// TIA Portal V19 export
// export: Created 2024-12-05T09:06:09.6853574Z, ExportSetting WithDefaults, DisplayName Totally Integrated Automation Portal, DisplayVersion V19 Update 1, DisplayName TIA Portal Openness, DisplayVersion V19 Update 1, DisplayName TIA Portal Version Control Interface, DisplayVersion V19, DisplayName SINAMICS Startdrive Advanced, DisplayVersion V19, DisplayName SINAMICS DCC, DisplayVersion V19, DisplayName SINAMICS Startdrive G130, G150, S120, S150, SINAMICS MV, G220, S200, S210, DisplayVersion V19, DisplayName SINAMICS Startdrive G110M, G120, G120C, G120D, G120P, G115D, DisplayVersion V19, DisplayName STEP 7 Professional, DisplayVersion V19 Update 1, DisplayName STEP 7 Safety, DisplayVersion V19 Update 1, DisplayName WinCC Advanced, DisplayVersion V19 Update 1, DisplayName WinCC Advanced / Unified PC, DisplayVersion V19 Update 1
DATA_BLOCK "GLOBAL"   // DB9
{ S7_Optimized_Access := 'TRUE' }
VERSION : 0.1
// stored: AutoNumber true, DBAccessibleFromOPCUA true, DBAccessibleFromWebserver true, InstanceOfName EM_GLOBAL, InstanceOfType UDT, IsOnlyStoredInLoadMemory false, IsWriteProtectedInAS false
"EM_GLOBAL"
   // VAR
   //    Gen : "GLOBAL_Gen";
   //    Param : "GLOBAL_Param";
   //    Recipe : "GLOBAL_Recipe";
   //    AlmLong : "GLOBAL_Alm";
   //    AlmTypeFbkLong : "AlmType";
   //    AlmTypeOkLong : "AlmType";
   //    AlmCauseFbkLong : "AlmCause";
   //    AlmCauseOkLong : "AlmCause";
   //    AlmStructLong : "STD_ALM_STRUCT";
   //    AlmBannerFbkLong : "STD_ALM_BAN_FBK";
   //    AlmShort : "GLOBAL_Alm";
   //    AlmTypeFbkShort : "AlmType";
   //    AlmTypeOkShort : "AlmType";
   //    AlmCauseFbkShort : "AlmCause";
   //    AlmCauseOkShort : "AlmCause";
   //    AlmStructShort : "STD_ALM_STRUCT";
   //    AlmBannerFbkShort : "STD_ALM_BAN_FBK";
   //    Sign : "GLOBAL_Sign";
   //    SignStruct : "STD_SIGN_STRUCT";
   //    SignBannerFbk : "STD_SIGN_BAN_FBK";
   //    Input : "GLOBAL_Input";
   //    Output : "GLOBAL_Output";
   //    Ons : "GLOBAL_Ons";
   //    AirTreatment : "AirTreatment";
   //    Summ : "GLOBAL_Summary";
   //    LightSiren : "LightSiren_Module";
   //    ExchangeCmd : "Exchange_FromGlobal";
   //    ExchangeCmd_Switchboard : "Exchange_FromGlobal_Switchboard";
   //    Downstream : "Interface_Downstream";
   //    "MyStateDeviceCab&Field" : Array[0..1023] of Bool;
   //    DC_Bus_Converter1 : "ACT_DC_BUS";
   //    DC_Bus_Converter2 : "ACT_DC_BUS";
   //    DC_Bus_Converter3 : "ACT_DC_BUS";
   //    DC_Bus_Converter4 : "ACT_DC_BUS";
   // END_VAR
BEGIN
   Gen.PlannerGroupSync := TRUE;
   Gen.PwrDriveShortCondOK := TRUE;
   Gen.PwrDriveLongCondOK := TRUE;
   Gen.PwrDriveShortDone := TRUE;
   Gen.PwrDriveLongDone := TRUE;
   Gen.StationOutOfTime := TRUE;
   Gen.AllPlcsRun := TRUE;
   Gen.PwrDriveShortIndex := 8192;
   Gen.PwrDriveLongIndex := 8192;
   Gen.DayOfWeek := 5;
   Gen.PanelConnectionError := 64;
   Gen.FirstAlmID := -1;
   Gen.TimePIDexecution := 8.0;
   Gen.TON_ResetNewAlm.PT := T#5S;
   Gen.TON_ResetNewSign.PT := T#1S;
   Gen.TON_PlannerGroupSync.PT := T#2S;
   Gen.TON_PlannerGroupSync.ET := T#2S;
   Gen.TON_PlannerGroupSync.IN := TRUE;
   Gen.TON_PlannerGroupSync.Q := TRUE;
   Gen.TON_WaitSaveRecipeOnLine.PT := T#5S;
   Gen.TON_WaitLoadRecipeOnLine.PT := T#5S;
   Gen.TON_AirMissing_Gta1.PT := T#2S;
   Gen.TON_AirMissing_Gta2.PT := T#2S;
   Gen.TON_AirMissing_Gta3.PT := T#2S;
   Gen.TON_AirMissing_Gta4.PT := T#2S;
   Gen.TON_AirMissing_Gta4.ET := T#2S;
   Gen.TON_AirMissing_Gta4.IN := TRUE;
   Gen.TON_AirMissing_Gta4.Q := TRUE;
   Gen.TON_AirMissing_Gta5.PT := T#2S;
   Gen.TON_AirMissing_Gta5.ET := T#2S;
   Gen.TON_AirMissing_Gta5.IN := TRUE;
   Gen.TON_AirMissing_Gta5.Q := TRUE;
   Gen.TON_AirMissing_Gta6.PT := T#2S;
   Gen.TON_RecipeDownloadTimeout.PT := T#5S;
   Gen.TON_RecipeUploadTimeout.PT := T#5S;
   Gen.TON_RecipeMaintConfigDownloadTimeout.PT := T#5S;
   Gen.TON_RecipeMaintConfigUploadTimeout.PT := T#5S;
   Gen.TON_RecipeTotalizersDownloadTimeout.PT := T#5S;
   Gen.TON_RecipeTotalizersUploadTimeout.PT := T#5S;
   Gen.TOF_ResetButtonAuto.PT := T#1S;
   Gen.TOF_ResetButtonAuto.ET := T#1S;
   Gen.TOF_ResetButtonGlobal.PT := T#300MS;
   Gen.TOF_ResetButtonGlobal.ET := T#300MS;
   Gen.TOF_SirenEna.PT := T#5S;
   Gen.TOF_SirenEna.ET := T#5S;
   Gen.TON_LineEmpty.PT := T#2S;
   Recipe.MngByHmi := TRUE;
   Recipe.MaxNumber := 99;
   Recipe.Online.TOF_SaveDone.PT := T#1S;
   Recipe.Online.TOF_LoadDone.PT := T#1S;
   Recipe.Offline.TOF_SaveDone.PT := T#1S;
   Recipe.Offline.TOF_LoadDone.PT := T#1S;
   // AlmLong.ThSwitch."0" : GLOBAL.AlmLong.ThSwitch.0 > Circuit breaker power supply 1 (1PW100QA8)
   // AlmLong.ThSwitch."1" : GLOBAL.AlmLong.ThSwitch.1 > Circuit breaker power supply 2 (1PW100QA9)
   // AlmLong.ThSwitch."2" : GLOBAL.AlmLong.ThSwitch.2 > Circuit breaker series main power supply (1PW113)
   // AlmLong.ThSwitch."3" : GLOBAL.AlmLong.ThSwitch.3 > Circuit breaker series field power supply (1PW114)
   // AlmLong.ThSwitch."4" : GLOBAL.AlmLong.ThSwitch.4 > Circuit breaker series sinamics power supply (1PW113)
   // AlmLong.ThSwitch."5" : GLOBAL.AlmLong.ThSwitch.5 > Circuit breaker series valves power supply (1PW116)
   // AlmLong.ThSwitch."6" : GLOBAL.AlmLong.ThSwitch.6 > Circuit breaker series lamps power supply (1PW115)
   // AlmLong.ThSwitch."7" : GLOBAL.AlmLong.ThSwitch.7 > Main trip isolator unit faul (1PW6KA2)
   // AlmLong.ThSwitch."8" : GLOBAL.AlmLong.ThSwitch.8
   // AlmLong.ThSwitch."9" : GLOBAL.AlmLong.ThSwitch.9
   // AlmLong.ThSwitch."10" : GLOBAL.AlmLong.ThSwitch.10 > Circuit breaker series blocking cycle (1PW110)
   // AlmLong.ThSwitch."11" : GLOBAL.AlmLong.ThSwitch.11 > Loto disconnected (1PW11QA2)
   // AlmLong.ThSwitch."12" : GLOBAL.AlmLong.ThSwitch.12
   // AlmLong.ThSwitch."13" : GLOBAL.AlmLong.ThSwitch.13 > Circuit breakers series depositors (1PW110)
   // AlmLong.ThSwitch."14" : GLOBAL.AlmLong.ThSwitch.14
   // AlmLong.ThSwitch."15" : GLOBAL.AlmLong.ThSwitch.15
   // AlmLong.ThSwitch."16" : GLOBAL.AlmLong.ThSwitch.16
   // AlmLong.ThSwitch."17" : GLOBAL.AlmLong.ThSwitch.17
   // AlmLong.ThSwitch."18" : GLOBAL.AlmLong.ThSwitch.18
   // AlmLong.ThSwitch."19" : GLOBAL.AlmLong.ThSwitch.19
   // AlmLong.ThSwitch."20" : GLOBAL.AlmLong.ThSwitch.20
   // AlmLong.ThSwitch."21" : GLOBAL.AlmLong.ThSwitch.21
   // AlmLong.ThSwitch."22" : GLOBAL.AlmLong.ThSwitch.22
   // AlmLong.ThSwitch."23" : GLOBAL.AlmLong.ThSwitch.23
   // AlmLong.ThSwitch."24" : GLOBAL.AlmLong.ThSwitch.24
   // AlmLong.ThSwitch."25" : GLOBAL.AlmLong.ThSwitch.25
   // AlmLong.ThSwitch."26" : GLOBAL.AlmLong.ThSwitch.26
   // AlmLong.ThSwitch."27" : GLOBAL.AlmLong.ThSwitch.27
   // AlmLong.ThSwitch."28" : GLOBAL.AlmLong.ThSwitch.28
   // AlmLong.ThSwitch."29" : GLOBAL.AlmLong.ThSwitch.29
   // AlmLong.ThSwitch."30" : GLOBAL.AlmLong.ThSwitch.30
   // AlmLong.ThSwitch."31" : GLOBAL.AlmLong.ThSwitch.31
   // AlmLong.SafeComm."0" : GLOBAL.AlmLong.SafeComm.0
   // AlmLong.SafeComm."1" : GLOBAL.AlmLong.SafeComm.1
   // AlmLong.SafeComm."2" : GLOBAL.AlmLong.SafeComm.2 > Fault on ethernet module (1PLC200KF4)
   // AlmLong.SafeComm."3" : GLOBAL.AlmLong.SafeComm.3 > Fault on ethernet module (1PLC200KF4A)
   // AlmLong.SafeComm."4" : GLOBAL.AlmLong.SafeComm.4 > Fault on ethernet module (1PLC200KF5)
   // AlmLong.SafeComm."5" : GLOBAL.AlmLong.SafeComm.5
   // AlmLong.SafeComm."6" : GLOBAL.AlmLong.SafeComm.6
   // AlmLong.SafeComm."7" : GLOBAL.AlmLong.SafeComm.7 > Communication fault DP1
   // AlmLong.SafeComm."8" : GLOBAL.AlmLong.SafeComm.8 > Communication fault DP2
   // AlmLong.SafeComm."9" : GLOBAL.AlmLong.SafeComm.9 > Communication fault DP3
   // AlmLong.SafeComm."10" : GLOBAL.AlmLong.SafeComm.10 > Communication fault DP4
   // AlmLong.SafeComm."11" : GLOBAL.AlmLong.SafeComm.11
   // AlmLong.SafeComm."12" : GLOBAL.AlmLong.SafeComm.12
   // AlmLong.SafeComm."13" : GLOBAL.AlmLong.SafeComm.13
   // AlmLong.SafeComm."14" : GLOBAL.AlmLong.SafeComm.14
   // AlmLong.SafeComm."15" : GLOBAL.AlmLong.SafeComm.15 > Communication fault point_IO 1 (1PLC300KF3)
   // AlmLong.SafeComm."16" : GLOBAL.AlmLong.SafeComm.16 > Communication fault point_IO 2 (1PLC350KF3)
   // AlmLong.SafeComm."17" : GLOBAL.AlmLong.SafeComm.17 > Communication fault point_IO 3 (1PLC400KF3)
   // AlmLong.SafeComm."18" : GLOBAL.AlmLong.SafeComm.18
   // AlmLong.SafeComm."19" : GLOBAL.AlmLong.SafeComm.19
   // AlmLong.SafeComm."20" : GLOBAL.AlmLong.SafeComm.20
   // AlmLong.SafeComm."21" : GLOBAL.AlmLong.SafeComm.21
   // AlmLong.SafeComm."22" : GLOBAL.AlmLong.SafeComm.22
   // AlmLong.SafeComm."23" : GLOBAL.AlmLong.SafeComm.23
   // AlmLong.SafeComm."24" : GLOBAL.AlmLong.SafeComm.24
   // AlmLong.SafeComm."25" : GLOBAL.AlmLong.SafeComm.25
   // AlmLong.SafeComm."26" : GLOBAL.AlmLong.SafeComm.26
   // AlmLong.SafeComm."27" : GLOBAL.AlmLong.SafeComm.27
   // AlmLong.SafeComm."28" : GLOBAL.AlmLong.SafeComm.28
   // AlmLong.SafeComm."29" : GLOBAL.AlmLong.SafeComm.29
   // AlmLong.SafeComm."30" : GLOBAL.AlmLong.SafeComm.30
   // AlmLong.SafeComm."31" : GLOBAL.AlmLong.SafeComm.31
   // AlmLong.SafeEmg."0" : GLOBAL.AlmLong.SafeEmg.0 > Emergency pressed on cabinet (1PLC340SF2)
   // AlmLong.SafeEmg."1" : GLOBAL.AlmLong.SafeEmg.1
   // AlmLong.SafeEmg."2" : GLOBAL.AlmLong.SafeEmg.2
   // AlmLong.SafeEmg."3" : GLOBAL.AlmLong.SafeEmg.3
   // AlmLong.SafeEmg."4" : GLOBAL.AlmLong.SafeEmg.4
   // AlmLong.SafeEmg."5" : GLOBAL.AlmLong.SafeEmg.5
   // AlmLong.SafeEmg."6" : GLOBAL.AlmLong.SafeEmg.6
   // AlmLong.SafeEmg."7" : GLOBAL.AlmLong.SafeEmg.7
   // AlmLong.SafeEmg."8" : GLOBAL.AlmLong.SafeEmg.8
   // AlmLong.SafeEmg."9" : GLOBAL.AlmLong.SafeEmg.9
   // AlmLong.SafeEmg."10" : GLOBAL.AlmLong.SafeEmg.10
   // AlmLong.SafeEmg."11" : GLOBAL.AlmLong.SafeEmg.11
   // AlmLong.SafeEmg."12" : GLOBAL.AlmLong.SafeEmg.12
   // AlmLong.SafeEmg."13" : GLOBAL.AlmLong.SafeEmg.13
   // AlmLong.SafeEmg."14" : GLOBAL.AlmLong.SafeEmg.14
   // AlmLong.SafeEmg."15" : GLOBAL.AlmLong.SafeEmg.15
   // AlmLong.SafeEmg."16" : GLOBAL.AlmLong.SafeEmg.16 > Instruction fault emergency pressed on cabinet (1PLC340SF2)
   // AlmLong.SafeEmg."17" : GLOBAL.AlmLong.SafeEmg.17
   // AlmLong.SafeEmg."18" : GLOBAL.AlmLong.SafeEmg.18
   // AlmLong.SafeEmg."19" : GLOBAL.AlmLong.SafeEmg.19
   // AlmLong.SafeEmg."20" : GLOBAL.AlmLong.SafeEmg.20
   // AlmLong.SafeEmg."21" : GLOBAL.AlmLong.SafeEmg.21
   // AlmLong.SafeEmg."22" : GLOBAL.AlmLong.SafeEmg.22
   // AlmLong.SafeEmg."23" : GLOBAL.AlmLong.SafeEmg.23
   // AlmLong.SafeEmg."24" : GLOBAL.AlmLong.SafeEmg.24
   // AlmLong.SafeEmg."25" : GLOBAL.AlmLong.SafeEmg.25
   // AlmLong.SafeEmg."26" : GLOBAL.AlmLong.SafeEmg.26
   // AlmLong.SafeEmg."27" : GLOBAL.AlmLong.SafeEmg.27
   // AlmLong.SafeEmg."28" : GLOBAL.AlmLong.SafeEmg.28
   // AlmLong.SafeEmg."29" : GLOBAL.AlmLong.SafeEmg.29
   // AlmLong.SafeEmg."30" : GLOBAL.AlmLong.SafeEmg.30
   // AlmLong.SafeEmg."31" : GLOBAL.AlmLong.SafeEmg.31 > Moulding emergency series safety no ok
   // AlmLong.SafeGuards."0" : GLOBAL.AlmLong.SafeGuards.0
   // AlmLong.SafeGuards."1" : GLOBAL.AlmLong.SafeGuards.1
   // AlmLong.SafeGuards."2" : GLOBAL.AlmLong.SafeGuards.2
   // AlmLong.SafeGuards."3" : GLOBAL.AlmLong.SafeGuards.3
   // AlmLong.SafeGuards."4" : GLOBAL.AlmLong.SafeGuards.4
   // AlmLong.SafeGuards."5" : GLOBAL.AlmLong.SafeGuards.5
   // AlmLong.SafeGuards."6" : GLOBAL.AlmLong.SafeGuards.6
   // AlmLong.SafeGuards."7" : GLOBAL.AlmLong.SafeGuards.7
   // AlmLong.SafeGuards."8" : GLOBAL.AlmLong.SafeGuards.8
   // AlmLong.SafeGuards."9" : GLOBAL.AlmLong.SafeGuards.9
   // AlmLong.SafeGuards."10" : GLOBAL.AlmLong.SafeGuards.10
   // AlmLong.SafeGuards."11" : GLOBAL.AlmLong.SafeGuards.11
   // AlmLong.SafeGuards."12" : GLOBAL.AlmLong.SafeGuards.12
   // AlmLong.SafeGuards."13" : GLOBAL.AlmLong.SafeGuards.13
   // AlmLong.SafeGuards."14" : GLOBAL.AlmLong.SafeGuards.14
   // AlmLong.SafeGuards."15" : GLOBAL.AlmLong.SafeGuards.15
   // AlmLong.SafeGuards."16" : GLOBAL.AlmLong.SafeGuards.16 > Module fault (1PLC340KF1)
   // AlmLong.SafeGuards."17" : GLOBAL.AlmLong.SafeGuards.17 > Module fault (1PLC390KF1)
   // AlmLong.SafeGuards."18" : GLOBAL.AlmLong.SafeGuards.18 > Module fault (1PLC391KF1)
   // AlmLong.SafeGuards."19" : GLOBAL.AlmLong.SafeGuards.19 > Module fault (1PLC396KF1)
   // AlmLong.SafeGuards."20" : GLOBAL.AlmLong.SafeGuards.20 > Module fault (1PLC398KF1)
   // AlmLong.SafeGuards."21" : GLOBAL.AlmLong.SafeGuards.21
   // AlmLong.SafeGuards."22" : GLOBAL.AlmLong.SafeGuards.22
   // AlmLong.SafeGuards."23" : GLOBAL.AlmLong.SafeGuards.23
   // AlmLong.SafeGuards."24" : GLOBAL.AlmLong.SafeGuards.24
   // AlmLong.SafeGuards."25" : GLOBAL.AlmLong.SafeGuards.25
   // AlmLong.SafeGuards."26" : GLOBAL.AlmLong.SafeGuards.26
   // AlmLong.SafeGuards."27" : GLOBAL.AlmLong.SafeGuards.27
   // AlmLong.SafeGuards."28" : GLOBAL.AlmLong.SafeGuards.28
   // AlmLong.SafeGuards."29" : GLOBAL.AlmLong.SafeGuards.29
   // AlmLong.SafeGuards."30" : GLOBAL.AlmLong.SafeGuards.30
   // AlmLong.SafeGuards."31" : GLOBAL.AlmLong.SafeGuards.31
   // AlmLong.GtaAirGroup."0" : GLOBAL.AlmLong.GtaAirGroup.0 > Module or instruction fault GTA air group 1 (1FM371BP2,3)
   AlmLong.GtaAirGroup."1" := FALSE;   // GLOBAL.AlmLong.GtaAirGroup.1 > Group GTA 1 missing air (1FM330BP6)
   // AlmLong.GtaAirGroup."2" : GLOBAL.AlmLong.GtaAirGroup.2 > Module or instruction fault GTA air group 2 (3VV372BP2,3)
   // AlmLong.GtaAirGroup."3" : GLOBAL.AlmLong.GtaAirGroup.3 > Group GTA 2 missing air (3VV330BP5)
   // AlmLong.GtaAirGroup."4" : GLOBAL.AlmLong.GtaAirGroup.4 > Module or instruction fault GTA air group 3 (4VV372BP2,3)
   AlmLong.GtaAirGroup."5" := FALSE;   // GLOBAL.AlmLong.GtaAirGroup.5 > Group GTA 3 missing air (4VV330BP5)
   AlmLong.GtaAirGroup."6" := TRUE;   // GLOBAL.AlmLong.GtaAirGroup.6 > Module or instruction fault GTA air group 4 (1RD372BP2,3)
   AlmLong.GtaAirGroup."7" := TRUE;   // GLOBAL.AlmLong.GtaAirGroup.7 > Group GTA 4 missing air (1RD330BP5)
   // AlmLong.GtaAirGroup."8" : GLOBAL.AlmLong.GtaAirGroup.8 > Module or instruction fault GTA air group 5 (1RD472BP2,3)
   AlmLong.GtaAirGroup."9" := TRUE;   // GLOBAL.AlmLong.GtaAirGroup.9 > Group GTA 5 missing air (1RD430BP2)
   // AlmLong.GtaAirGroup."10" : GLOBAL.AlmLong.GtaAirGroup.10
   // AlmLong.GtaAirGroup."11" : GLOBAL.AlmLong.GtaAirGroup.11
   // AlmLong.GtaAirGroup."12" : GLOBAL.AlmLong.GtaAirGroup.12
   // AlmLong.GtaAirGroup."13" : GLOBAL.AlmLong.GtaAirGroup.13
   // AlmLong.GtaAirGroup."14" : GLOBAL.AlmLong.GtaAirGroup.14
   // AlmLong.GtaAirGroup."15" : GLOBAL.AlmLong.GtaAirGroup.15
   // AlmLong.GtaAirGroup."16" : GLOBAL.AlmLong.GtaAirGroup.16
   // AlmLong.GtaAirGroup."17" : GLOBAL.AlmLong.GtaAirGroup.17
   // AlmLong.GtaAirGroup."18" : GLOBAL.AlmLong.GtaAirGroup.18
   // AlmLong.GtaAirGroup."19" : GLOBAL.AlmLong.GtaAirGroup.19
   // AlmLong.GtaAirGroup."20" : GLOBAL.AlmLong.GtaAirGroup.20
   // AlmLong.GtaAirGroup."21" : GLOBAL.AlmLong.GtaAirGroup.21
   // AlmLong.GtaAirGroup."22" : GLOBAL.AlmLong.GtaAirGroup.22
   // AlmLong.GtaAirGroup."23" : GLOBAL.AlmLong.GtaAirGroup.23
   // AlmLong.GtaAirGroup."24" : GLOBAL.AlmLong.GtaAirGroup.24
   // AlmLong.GtaAirGroup."25" : GLOBAL.AlmLong.GtaAirGroup.25
   // AlmLong.GtaAirGroup."26" : GLOBAL.AlmLong.GtaAirGroup.26
   // AlmLong.GtaAirGroup."27" : GLOBAL.AlmLong.GtaAirGroup.27
   // AlmLong.GtaAirGroup."28" : GLOBAL.AlmLong.GtaAirGroup.28
   // AlmLong.GtaAirGroup."29" : GLOBAL.AlmLong.GtaAirGroup.29
   // AlmLong.GtaAirGroup."30" : GLOBAL.AlmLong.GtaAirGroup.30
   // AlmLong.GtaAirGroup."31" : GLOBAL.AlmLong.GtaAirGroup.31
   // AlmLong.Major."0" : GLOBAL.AlmLong.Major.0 > Module or instruction fault emergency + carter feedback (1CH130KF2)
   // AlmLong.Major."1" : GLOBAL.AlmLong.Major.1 > Module or instruction fault feedback emergency (1CH130KF4)
   // AlmLong.Major."2" : GLOBAL.AlmLong.Major.2 > Module or instruction fault feedback emergency (1CH130KF6)
   // AlmLong.Major."3" : GLOBAL.AlmLong.Major.3 > Module or instruction fault feedback fans emergency contactor branch 2
   // AlmLong.Major."4" : GLOBAL.AlmLong.Major.4
   // AlmLong.Major."5" : GLOBAL.AlmLong.Major.5 > Module or instruction fault feedback emergency + carter branch 1 (1CH132KF2)
   // AlmLong.Major."6" : GLOBAL.AlmLong.Major.6 > Module or instruction fault feedback emergency + carter branch 2 (1CH132KF4)
   // AlmLong.Major."7" : GLOBAL.AlmLong.Major.7
   // AlmLong.Major."8" : GLOBAL.AlmLong.Major.8
   // AlmLong.Major."9" : GLOBAL.AlmLong.Major.9
   // AlmLong.Major."10" : GLOBAL.AlmLong.Major.10
   // AlmLong.Major."11" : GLOBAL.AlmLong.Major.11
   // AlmLong.Major."12" : GLOBAL.AlmLong.Major.12
   // AlmLong.Major."13" : GLOBAL.AlmLong.Major.13
   // AlmLong.Major."14" : GLOBAL.AlmLong.Major.14
   // AlmLong.Major."15" : GLOBAL.AlmLong.Major.15 > Presence 24Vdc supply
   // AlmLong.Major."16" : GLOBAL.AlmLong.Major.16
   // AlmLong.Major."17" : GLOBAL.AlmLong.Major.17
   // AlmLong.Major."18" : GLOBAL.AlmLong.Major.18
   // AlmLong.Major."19" : GLOBAL.AlmLong.Major.19
   // AlmLong.Major."20" : GLOBAL.AlmLong.Major.20 > Dc bus converter 1 fault
   // AlmLong.Major."21" : GLOBAL.AlmLong.Major.21 > Dc bus converter 2 fault
   // AlmLong.Major."22" : GLOBAL.AlmLong.Major.22 > Dc bus converter 3 fault
   // AlmLong.Major."23" : GLOBAL.AlmLong.Major.23 > Dc bus converter 4 fault
   // AlmLong.Major."24" : GLOBAL.AlmLong.Major.24
   // AlmLong.Major."25" : GLOBAL.AlmLong.Major.25
   // AlmLong.Major."26" : GLOBAL.AlmLong.Major.26
   // AlmLong.Major."27" : GLOBAL.AlmLong.Major.27
   // AlmLong.Major."28" : GLOBAL.AlmLong.Major.28
   // AlmLong.Major."29" : GLOBAL.AlmLong.Major.29
   // AlmLong.Major."30" : GLOBAL.AlmLong.Major.30
   // AlmLong.Major."31" : GLOBAL.AlmLong.Major.31
   // AlmLong.Minor."0" : GLOBAL.AlmLong.Minor.0 > Connection HMI server error
   // AlmLong.Minor."1" : GLOBAL.AlmLong.Minor.1 > Request update parameters from PLC to HMI
   // AlmLong.Minor."2" : GLOBAL.AlmLong.Minor.2 > Recipe download from HMI error
   // AlmLong.Minor."3" : GLOBAL.AlmLong.Minor.3 > Request maintenance configuration from PLC to HMI
   // AlmLong.Minor."4" : GLOBAL.AlmLong.Minor.4 > Recipe maintenance configuration download from HMI error
   // AlmLong.Minor."5" : GLOBAL.AlmLong.Minor.5 > Request update totalizers from PLC to HMI
   // AlmLong.Minor."6" : GLOBAL.AlmLong.Minor.6 > Recipe totalizers download from HMI error
   // AlmLong.Minor."7" : GLOBAL.AlmLong.Minor.7
   // AlmLong.Minor."8" : GLOBAL.AlmLong.Minor.8 > More then one drum enabled, they will be reset
   // AlmLong.Minor."9" : GLOBAL.AlmLong.Minor.9
   // AlmLong.Minor."10" : GLOBAL.AlmLong.Minor.10
   // AlmLong.Minor."11" : GLOBAL.AlmLong.Minor.11
   // AlmLong.Minor."12" : GLOBAL.AlmLong.Minor.12
   // AlmLong.Minor."13" : GLOBAL.AlmLong.Minor.13
   // AlmLong.Minor."14" : GLOBAL.AlmLong.Minor.14
   // AlmLong.Minor."15" : GLOBAL.AlmLong.Minor.15 > Downstream communication fault
   // AlmLong.Minor."16" : GLOBAL.AlmLong.Minor.16
   // AlmLong.Minor."17" : GLOBAL.AlmLong.Minor.17
   // AlmLong.Minor."18" : GLOBAL.AlmLong.Minor.18
   // AlmLong.Minor."19" : GLOBAL.AlmLong.Minor.19
   // AlmLong.Minor."20" : GLOBAL.AlmLong.Minor.20
   // AlmLong.Minor."21" : GLOBAL.AlmLong.Minor.21
   // AlmLong.Minor."22" : GLOBAL.AlmLong.Minor.22
   // AlmLong.Minor."23" : GLOBAL.AlmLong.Minor.23
   // AlmLong.Minor."24" : GLOBAL.AlmLong.Minor.24
   // AlmLong.Minor."25" : GLOBAL.AlmLong.Minor.25
   // AlmLong.Minor."26" : GLOBAL.AlmLong.Minor.26
   // AlmLong.Minor."27" : GLOBAL.AlmLong.Minor.27
   // AlmLong.Minor."28" : GLOBAL.AlmLong.Minor.28
   // AlmLong.Minor."29" : GLOBAL.AlmLong.Minor.29
   // AlmLong.Minor."30" : GLOBAL.AlmLong.Minor.30
   // AlmLong.Minor."31" : GLOBAL.AlmLong.Minor.31
   AlmTypeFbkLong.GtaAirGroup := TRUE;
   AlmTypeOkLong.ThSwitch := TRUE;
   AlmTypeOkLong.SafeComm := TRUE;
   AlmTypeOkLong.SafeEmg := TRUE;
   AlmTypeOkLong.SafeGuards := TRUE;
   AlmTypeOkLong.GtaAirGroup := FALSE;
   AlmTypeOkLong.Major := TRUE;
   AlmTypeOkLong.Minor := TRUE;
   AlmTypeOkLong.Spare07 := TRUE;
   AlmTypeOkLong.Spare08 := TRUE;
   AlmTypeOkLong.Spare09 := TRUE;
   AlmTypeOkLong.Spare10 := TRUE;
   AlmTypeOkLong.Spare11 := TRUE;
   AlmTypeOkLong.Spare12 := TRUE;
   AlmTypeOkLong.Spare13 := TRUE;
   AlmTypeOkLong.Spare14 := TRUE;
   AlmTypeOkLong.Spare15 := TRUE;
   AlmTypeOkLong.Spare16 := TRUE;
   AlmTypeOkLong.Spare17 := TRUE;
   AlmTypeOkLong.Spare18 := TRUE;
   AlmTypeOkLong.Spare19 := TRUE;
   AlmTypeOkLong.Spare20 := TRUE;
   AlmTypeOkLong.Spare21 := TRUE;
   AlmTypeOkLong.Spare22 := TRUE;
   AlmTypeOkLong.Spare23 := TRUE;
   AlmTypeOkLong.Spare24 := TRUE;
   AlmTypeOkLong.Spare25 := TRUE;
   AlmTypeOkLong.Spare26 := TRUE;
   AlmTypeOkLong.Spare27 := TRUE;
   AlmTypeOkLong.Spare28 := TRUE;
   AlmTypeOkLong.Spare29 := TRUE;
   AlmTypeOkLong.Spare30 := TRUE;
   AlmTypeOkLong.Spare31 := TRUE;
   AlmCauseFbkLong.Ext := TRUE;
   AlmCauseOkLong.Ope := TRUE;
   AlmCauseOkLong.Ust := TRUE;
   AlmCauseOkLong.Dst := TRUE;
   AlmCauseOkLong.Ext := FALSE;
   AlmCauseOkLong.Mac := TRUE;
   AlmCauseOkLong.Spare05 := TRUE;
   AlmCauseOkLong.Spare06 := TRUE;
   AlmCauseOkLong.Spare07 := TRUE;
   AlmCauseOkLong.Spare08 := TRUE;
   AlmCauseOkLong.Spare09 := TRUE;
   AlmCauseOkLong.Spare10 := TRUE;
   AlmCauseOkLong.Spare11 := TRUE;
   AlmCauseOkLong.Spare12 := TRUE;
   AlmCauseOkLong.Spare13 := TRUE;
   AlmCauseOkLong.Spare14 := TRUE;
   AlmCauseOkLong.Spare15 := TRUE;
   AlmCauseOkLong.Spare16 := TRUE;
   AlmCauseOkLong.Spare17 := TRUE;
   AlmCauseOkLong.Spare18 := TRUE;
   AlmCauseOkLong.Spare19 := TRUE;
   AlmCauseOkLong.Spare20 := TRUE;
   AlmCauseOkLong.Spare21 := TRUE;
   AlmCauseOkLong.Spare22 := TRUE;
   AlmCauseOkLong.Spare23 := TRUE;
   AlmCauseOkLong.Spare24 := TRUE;
   AlmCauseOkLong.Spare25 := TRUE;
   AlmCauseOkLong.Spare26 := TRUE;
   AlmCauseOkLong.Spare27 := TRUE;
   AlmCauseOkLong.Spare28 := TRUE;
   AlmCauseOkLong.Spare29 := TRUE;
   AlmCauseOkLong.Spare30 := TRUE;
   AlmCauseOkLong.Spare31 := TRUE;
   AlmStructLong.Alm[4] := 704;
   AlmStructLong.Category[32..63] := 1;
   AlmStructLong.Category[64..95] := 2;
   AlmStructLong.Category[96..127] := 3;
   AlmStructLong.Category[128..159] := 4;
   AlmStructLong.Category[160..191] := 5;
   AlmStructLong.Category[192..1023] := 6;
   AlmStructLong.BannerPriority[32..63] := 1;
   AlmStructLong.BannerPriority[64..95] := 2;
   AlmStructLong.BannerPriority[96..127] := 3;
   AlmStructLong.BannerPriority[128..159] := 4;
   AlmStructLong.BannerPriority[160..191] := 5;
   AlmStructLong.BannerPriority[192..1023] := 6;
   AlmStructLong.Cause[0..63] := 4;
   AlmStructLong.Cause[128..159] := 3;
   AlmStructLong.Cause[160..1023] := 4;
   AlmBannerFbkLong.AlmPriority := 4;
   AlmBannerFbkLong.AlmCategory := 4;
   AlmBannerFbkLong.AlmCause := 3;
   AlmBannerFbkLong.AlmID := 640134;
   // AlmShort.ThSwitch."0" : GLOBAL.AlmShort.ThSwitch.0
   // AlmShort.ThSwitch."1" : GLOBAL.AlmShort.ThSwitch.1
   // AlmShort.ThSwitch."2" : GLOBAL.AlmShort.ThSwitch.2
   // AlmShort.ThSwitch."3" : GLOBAL.AlmShort.ThSwitch.3
   // AlmShort.ThSwitch."4" : GLOBAL.AlmShort.ThSwitch.4
   // AlmShort.ThSwitch."5" : GLOBAL.AlmShort.ThSwitch.5
   // AlmShort.ThSwitch."6" : GLOBAL.AlmShort.ThSwitch.6
   // AlmShort.ThSwitch."7" : GLOBAL.AlmShort.ThSwitch.7
   // AlmShort.ThSwitch."8" : GLOBAL.AlmShort.ThSwitch.8
   // AlmShort.ThSwitch."9" : GLOBAL.AlmShort.ThSwitch.9
   // AlmShort.ThSwitch."10" : GLOBAL.AlmShort.ThSwitch.10
   // AlmShort.ThSwitch."11" : GLOBAL.AlmShort.ThSwitch.11
   // AlmShort.ThSwitch."12" : GLOBAL.AlmShort.ThSwitch.12
   // AlmShort.ThSwitch."13" : GLOBAL.AlmShort.ThSwitch.13
   // AlmShort.ThSwitch."14" : GLOBAL.AlmShort.ThSwitch.14
   // AlmShort.ThSwitch."15" : GLOBAL.AlmShort.ThSwitch.15
   // AlmShort.ThSwitch."16" : GLOBAL.AlmShort.ThSwitch.16
   // AlmShort.ThSwitch."17" : GLOBAL.AlmShort.ThSwitch.17
   // AlmShort.ThSwitch."18" : GLOBAL.AlmShort.ThSwitch.18
   // AlmShort.ThSwitch."19" : GLOBAL.AlmShort.ThSwitch.19
   // AlmShort.ThSwitch."20" : GLOBAL.AlmShort.ThSwitch.20
   // AlmShort.ThSwitch."21" : GLOBAL.AlmShort.ThSwitch.21
   // AlmShort.ThSwitch."22" : GLOBAL.AlmShort.ThSwitch.22
   // AlmShort.ThSwitch."23" : GLOBAL.AlmShort.ThSwitch.23
   // AlmShort.ThSwitch."24" : GLOBAL.AlmShort.ThSwitch.24
   // AlmShort.ThSwitch."25" : GLOBAL.AlmShort.ThSwitch.25
   // AlmShort.ThSwitch."26" : GLOBAL.AlmShort.ThSwitch.26
   // AlmShort.ThSwitch."27" : GLOBAL.AlmShort.ThSwitch.27
   // AlmShort.ThSwitch."28" : GLOBAL.AlmShort.ThSwitch.28
   // AlmShort.ThSwitch."29" : GLOBAL.AlmShort.ThSwitch.29
   // AlmShort.ThSwitch."30" : GLOBAL.AlmShort.ThSwitch.30
   // AlmShort.ThSwitch."31" : GLOBAL.AlmShort.ThSwitch.31
   // AlmShort.SafeComm."0" : GLOBAL.AlmShort.SafeComm.0
   // AlmShort.SafeComm."1" : GLOBAL.AlmShort.SafeComm.1
   // AlmShort.SafeComm."2" : GLOBAL.AlmShort.SafeComm.2
   // AlmShort.SafeComm."3" : GLOBAL.AlmShort.SafeComm.3
   // AlmShort.SafeComm."4" : GLOBAL.AlmShort.SafeComm.4
   // AlmShort.SafeComm."5" : GLOBAL.AlmShort.SafeComm.5
   // AlmShort.SafeComm."6" : GLOBAL.AlmShort.SafeComm.6
   // AlmShort.SafeComm."7" : GLOBAL.AlmShort.SafeComm.7
   // AlmShort.SafeComm."8" : GLOBAL.AlmShort.SafeComm.8
   // AlmShort.SafeComm."9" : GLOBAL.AlmShort.SafeComm.9
   // AlmShort.SafeComm."10" : GLOBAL.AlmShort.SafeComm.10
   // AlmShort.SafeComm."11" : GLOBAL.AlmShort.SafeComm.11
   // AlmShort.SafeComm."12" : GLOBAL.AlmShort.SafeComm.12
   // AlmShort.SafeComm."13" : GLOBAL.AlmShort.SafeComm.13
   // AlmShort.SafeComm."14" : GLOBAL.AlmShort.SafeComm.14
   // AlmShort.SafeComm."15" : GLOBAL.AlmShort.SafeComm.15
   // AlmShort.SafeComm."16" : GLOBAL.AlmShort.SafeComm.16
   // AlmShort.SafeComm."17" : GLOBAL.AlmShort.SafeComm.17
   // AlmShort.SafeComm."18" : GLOBAL.AlmShort.SafeComm.18
   // AlmShort.SafeComm."19" : GLOBAL.AlmShort.SafeComm.19
   // AlmShort.SafeComm."20" : GLOBAL.AlmShort.SafeComm.20
   // AlmShort.SafeComm."21" : GLOBAL.AlmShort.SafeComm.21
   // AlmShort.SafeComm."22" : GLOBAL.AlmShort.SafeComm.22
   // AlmShort.SafeComm."23" : GLOBAL.AlmShort.SafeComm.23
   // AlmShort.SafeComm."24" : GLOBAL.AlmShort.SafeComm.24
   // AlmShort.SafeComm."25" : GLOBAL.AlmShort.SafeComm.25
   // AlmShort.SafeComm."26" : GLOBAL.AlmShort.SafeComm.26
   // AlmShort.SafeComm."27" : GLOBAL.AlmShort.SafeComm.27
   // AlmShort.SafeComm."28" : GLOBAL.AlmShort.SafeComm.28
   // AlmShort.SafeComm."29" : GLOBAL.AlmShort.SafeComm.29
   // AlmShort.SafeComm."30" : GLOBAL.AlmShort.SafeComm.30
   // AlmShort.SafeComm."31" : GLOBAL.AlmShort.SafeComm.31
   // AlmShort.SafeEmg."0" : GLOBAL.AlmShort.SafeEmg.0
   // AlmShort.SafeEmg."1" : GLOBAL.AlmShort.SafeEmg.1 >
   // AlmShort.SafeEmg."2" : GLOBAL.AlmShort.SafeEmg.2
   // AlmShort.SafeEmg."3" : GLOBAL.AlmShort.SafeEmg.3
   // AlmShort.SafeEmg."4" : GLOBAL.AlmShort.SafeEmg.4
   // AlmShort.SafeEmg."5" : GLOBAL.AlmShort.SafeEmg.5
   // AlmShort.SafeEmg."6" : GLOBAL.AlmShort.SafeEmg.6
   // AlmShort.SafeEmg."7" : GLOBAL.AlmShort.SafeEmg.7
   // AlmShort.SafeEmg."8" : GLOBAL.AlmShort.SafeEmg.8
   // AlmShort.SafeEmg."9" : GLOBAL.AlmShort.SafeEmg.9
   // AlmShort.SafeEmg."10" : GLOBAL.AlmShort.SafeEmg.10
   // AlmShort.SafeEmg."11" : GLOBAL.AlmShort.SafeEmg.11
   // AlmShort.SafeEmg."12" : GLOBAL.AlmShort.SafeEmg.12
   // AlmShort.SafeEmg."13" : GLOBAL.AlmShort.SafeEmg.13
   // AlmShort.SafeEmg."14" : GLOBAL.AlmShort.SafeEmg.14
   // AlmShort.SafeEmg."15" : GLOBAL.AlmShort.SafeEmg.15
   // AlmShort.SafeEmg."16" : GLOBAL.AlmShort.SafeEmg.16
   // AlmShort.SafeEmg."17" : GLOBAL.AlmShort.SafeEmg.17
   // AlmShort.SafeEmg."18" : GLOBAL.AlmShort.SafeEmg.18
   // AlmShort.SafeEmg."19" : GLOBAL.AlmShort.SafeEmg.19
   // AlmShort.SafeEmg."20" : GLOBAL.AlmShort.SafeEmg.20
   // AlmShort.SafeEmg."21" : GLOBAL.AlmShort.SafeEmg.21
   // AlmShort.SafeEmg."22" : GLOBAL.AlmShort.SafeEmg.22
   // AlmShort.SafeEmg."23" : GLOBAL.AlmShort.SafeEmg.23
   // AlmShort.SafeEmg."24" : GLOBAL.AlmShort.SafeEmg.24
   // AlmShort.SafeEmg."25" : GLOBAL.AlmShort.SafeEmg.25
   // AlmShort.SafeEmg."26" : GLOBAL.AlmShort.SafeEmg.26
   // AlmShort.SafeEmg."27" : GLOBAL.AlmShort.SafeEmg.27
   // AlmShort.SafeEmg."28" : GLOBAL.AlmShort.SafeEmg.28
   // AlmShort.SafeEmg."29" : GLOBAL.AlmShort.SafeEmg.29
   // AlmShort.SafeEmg."30" : GLOBAL.AlmShort.SafeEmg.30
   // AlmShort.SafeEmg."31" : GLOBAL.AlmShort.SafeEmg.31
   // AlmShort.SafeGuards."0" : GLOBAL.AlmShort.SafeGuards.0
   // AlmShort.SafeGuards."1" : GLOBAL.AlmShort.SafeGuards.1
   // AlmShort.SafeGuards."2" : GLOBAL.AlmShort.SafeGuards.2
   // AlmShort.SafeGuards."3" : GLOBAL.AlmShort.SafeGuards.3
   // AlmShort.SafeGuards."4" : GLOBAL.AlmShort.SafeGuards.4
   // AlmShort.SafeGuards."5" : GLOBAL.AlmShort.SafeGuards.5
   // AlmShort.SafeGuards."6" : GLOBAL.AlmShort.SafeGuards.6
   // AlmShort.SafeGuards."7" : GLOBAL.AlmShort.SafeGuards.7
   // AlmShort.SafeGuards."8" : GLOBAL.AlmShort.SafeGuards.8
   // AlmShort.SafeGuards."9" : GLOBAL.AlmShort.SafeGuards.9
   // AlmShort.SafeGuards."10" : GLOBAL.AlmShort.SafeGuards.10
   // AlmShort.SafeGuards."11" : GLOBAL.AlmShort.SafeGuards.11
   // AlmShort.SafeGuards."12" : GLOBAL.AlmShort.SafeGuards.12
   // AlmShort.SafeGuards."13" : GLOBAL.AlmShort.SafeGuards.13
   // AlmShort.SafeGuards."14" : GLOBAL.AlmShort.SafeGuards.14
   // AlmShort.SafeGuards."15" : GLOBAL.AlmShort.SafeGuards.15
   // AlmShort.SafeGuards."16" : GLOBAL.AlmShort.SafeGuards.16
   // AlmShort.SafeGuards."17" : GLOBAL.AlmShort.SafeGuards.17
   // AlmShort.SafeGuards."18" : GLOBAL.AlmShort.SafeGuards.18
   // AlmShort.SafeGuards."19" : GLOBAL.AlmShort.SafeGuards.19
   // AlmShort.SafeGuards."20" : GLOBAL.AlmShort.SafeGuards.20
   // AlmShort.SafeGuards."21" : GLOBAL.AlmShort.SafeGuards.21
   // AlmShort.SafeGuards."22" : GLOBAL.AlmShort.SafeGuards.22
   // AlmShort.SafeGuards."23" : GLOBAL.AlmShort.SafeGuards.23
   // AlmShort.SafeGuards."24" : GLOBAL.AlmShort.SafeGuards.24
   // AlmShort.SafeGuards."25" : GLOBAL.AlmShort.SafeGuards.25
   // AlmShort.SafeGuards."26" : GLOBAL.AlmShort.SafeGuards.26
   // AlmShort.SafeGuards."27" : GLOBAL.AlmShort.SafeGuards.27
   // AlmShort.SafeGuards."28" : GLOBAL.AlmShort.SafeGuards.28
   // AlmShort.SafeGuards."29" : GLOBAL.AlmShort.SafeGuards.29
   // AlmShort.SafeGuards."30" : GLOBAL.AlmShort.SafeGuards.30
   // AlmShort.SafeGuards."31" : GLOBAL.AlmShort.SafeGuards.31
   // AlmShort.GtaAirGroup."0" : GLOBAL.AlmShort.GtaAirGroup.0
   // AlmShort.GtaAirGroup."1" : GLOBAL.AlmShort.GtaAirGroup.1
   // AlmShort.GtaAirGroup."2" : GLOBAL.AlmShort.GtaAirGroup.2
   // AlmShort.GtaAirGroup."3" : GLOBAL.AlmShort.GtaAirGroup.3
   // AlmShort.GtaAirGroup."4" : GLOBAL.AlmShort.GtaAirGroup.4
   // AlmShort.GtaAirGroup."5" : GLOBAL.AlmShort.GtaAirGroup.5
   // AlmShort.GtaAirGroup."6" : GLOBAL.AlmShort.GtaAirGroup.6
   // AlmShort.GtaAirGroup."7" : GLOBAL.AlmShort.GtaAirGroup.7
   // AlmShort.GtaAirGroup."8" : GLOBAL.AlmShort.GtaAirGroup.8
   // AlmShort.GtaAirGroup."9" : GLOBAL.AlmShort.GtaAirGroup.9
   // AlmShort.GtaAirGroup."10" : GLOBAL.AlmShort.GtaAirGroup.10
   // AlmShort.GtaAirGroup."11" : GLOBAL.AlmShort.GtaAirGroup.11
   // AlmShort.GtaAirGroup."12" : GLOBAL.AlmShort.GtaAirGroup.12
   // AlmShort.GtaAirGroup."13" : GLOBAL.AlmShort.GtaAirGroup.13
   // AlmShort.GtaAirGroup."14" : GLOBAL.AlmShort.GtaAirGroup.14
   // AlmShort.GtaAirGroup."15" : GLOBAL.AlmShort.GtaAirGroup.15
   // AlmShort.GtaAirGroup."16" : GLOBAL.AlmShort.GtaAirGroup.16
   // AlmShort.GtaAirGroup."17" : GLOBAL.AlmShort.GtaAirGroup.17
   // AlmShort.GtaAirGroup."18" : GLOBAL.AlmShort.GtaAirGroup.18
   // AlmShort.GtaAirGroup."19" : GLOBAL.AlmShort.GtaAirGroup.19
   // AlmShort.GtaAirGroup."20" : GLOBAL.AlmShort.GtaAirGroup.20
   // AlmShort.GtaAirGroup."21" : GLOBAL.AlmShort.GtaAirGroup.21
   // AlmShort.GtaAirGroup."22" : GLOBAL.AlmShort.GtaAirGroup.22
   // AlmShort.GtaAirGroup."23" : GLOBAL.AlmShort.GtaAirGroup.23
   // AlmShort.GtaAirGroup."24" : GLOBAL.AlmShort.GtaAirGroup.24
   // AlmShort.GtaAirGroup."25" : GLOBAL.AlmShort.GtaAirGroup.25
   // AlmShort.GtaAirGroup."26" : GLOBAL.AlmShort.GtaAirGroup.26
   // AlmShort.GtaAirGroup."27" : GLOBAL.AlmShort.GtaAirGroup.27
   // AlmShort.GtaAirGroup."28" : GLOBAL.AlmShort.GtaAirGroup.28
   // AlmShort.GtaAirGroup."29" : GLOBAL.AlmShort.GtaAirGroup.29
   // AlmShort.GtaAirGroup."30" : GLOBAL.AlmShort.GtaAirGroup.30
   // AlmShort.GtaAirGroup."31" : GLOBAL.AlmShort.GtaAirGroup.31
   // AlmShort.Major."0" : GLOBAL.AlmShort.Major.0
   // AlmShort.Major."1" : GLOBAL.AlmShort.Major.1
   // AlmShort.Major."2" : GLOBAL.AlmShort.Major.2
   // AlmShort.Major."3" : GLOBAL.AlmShort.Major.3
   // AlmShort.Major."4" : GLOBAL.AlmShort.Major.4
   // AlmShort.Major."5" : GLOBAL.AlmShort.Major.5
   // AlmShort.Major."6" : GLOBAL.AlmShort.Major.6
   // AlmShort.Major."7" : GLOBAL.AlmShort.Major.7
   // AlmShort.Major."8" : GLOBAL.AlmShort.Major.8
   // AlmShort.Major."9" : GLOBAL.AlmShort.Major.9
   // AlmShort.Major."10" : GLOBAL.AlmShort.Major.10
   // AlmShort.Major."11" : GLOBAL.AlmShort.Major.11
   // AlmShort.Major."12" : GLOBAL.AlmShort.Major.12
   // AlmShort.Major."13" : GLOBAL.AlmShort.Major.13
   // AlmShort.Major."14" : GLOBAL.AlmShort.Major.14
   // AlmShort.Major."15" : GLOBAL.AlmShort.Major.15
   // AlmShort.Major."16" : GLOBAL.AlmShort.Major.16
   // AlmShort.Major."17" : GLOBAL.AlmShort.Major.17
   // AlmShort.Major."18" : GLOBAL.AlmShort.Major.18
   // AlmShort.Major."19" : GLOBAL.AlmShort.Major.19
   // AlmShort.Major."20" : GLOBAL.AlmShort.Major.20
   // AlmShort.Major."21" : GLOBAL.AlmShort.Major.21
   // AlmShort.Major."22" : GLOBAL.AlmShort.Major.22
   // AlmShort.Major."23" : GLOBAL.AlmShort.Major.23
   // AlmShort.Major."24" : GLOBAL.AlmShort.Major.24
   // AlmShort.Major."25" : GLOBAL.AlmShort.Major.25
   // AlmShort.Major."26" : GLOBAL.AlmShort.Major.26
   // AlmShort.Major."27" : GLOBAL.AlmShort.Major.27
   // AlmShort.Major."28" : GLOBAL.AlmShort.Major.28
   // AlmShort.Major."29" : GLOBAL.AlmShort.Major.29
   // AlmShort.Major."30" : GLOBAL.AlmShort.Major.30
   // AlmShort.Major."31" : GLOBAL.AlmShort.Major.31
   // AlmShort.Minor."0" : GLOBAL.AlmShort.Minor.0
   // AlmShort.Minor."1" : GLOBAL.AlmShort.Minor.1
   // AlmShort.Minor."2" : GLOBAL.AlmShort.Minor.2
   // AlmShort.Minor."3" : GLOBAL.AlmShort.Minor.3
   // AlmShort.Minor."4" : GLOBAL.AlmShort.Minor.4
   // AlmShort.Minor."5" : GLOBAL.AlmShort.Minor.5
   // AlmShort.Minor."6" : GLOBAL.AlmShort.Minor.6
   // AlmShort.Minor."7" : GLOBAL.AlmShort.Minor.7
   // AlmShort.Minor."8" : GLOBAL.AlmShort.Minor.8
   // AlmShort.Minor."9" : GLOBAL.AlmShort.Minor.9
   // AlmShort.Minor."10" : GLOBAL.AlmShort.Minor.10
   // AlmShort.Minor."11" : GLOBAL.AlmShort.Minor.11
   // AlmShort.Minor."12" : GLOBAL.AlmShort.Minor.12
   // AlmShort.Minor."13" : GLOBAL.AlmShort.Minor.13
   // AlmShort.Minor."14" : GLOBAL.AlmShort.Minor.14
   // AlmShort.Minor."15" : GLOBAL.AlmShort.Minor.15
   // AlmShort.Minor."16" : GLOBAL.AlmShort.Minor.16
   // AlmShort.Minor."17" : GLOBAL.AlmShort.Minor.17
   // AlmShort.Minor."18" : GLOBAL.AlmShort.Minor.18
   // AlmShort.Minor."19" : GLOBAL.AlmShort.Minor.19
   // AlmShort.Minor."20" : GLOBAL.AlmShort.Minor.20
   // AlmShort.Minor."21" : GLOBAL.AlmShort.Minor.21
   // AlmShort.Minor."22" : GLOBAL.AlmShort.Minor.22
   // AlmShort.Minor."23" : GLOBAL.AlmShort.Minor.23
   // AlmShort.Minor."24" : GLOBAL.AlmShort.Minor.24
   // AlmShort.Minor."25" : GLOBAL.AlmShort.Minor.25
   // AlmShort.Minor."26" : GLOBAL.AlmShort.Minor.26
   // AlmShort.Minor."27" : GLOBAL.AlmShort.Minor.27
   // AlmShort.Minor."28" : GLOBAL.AlmShort.Minor.28
   // AlmShort.Minor."29" : GLOBAL.AlmShort.Minor.29
   // AlmShort.Minor."30" : GLOBAL.AlmShort.Minor.30
   // AlmShort.Minor."31" : GLOBAL.AlmShort.Minor.31
   AlmTypeOkShort.ThSwitch := TRUE;
   AlmTypeOkShort.SafeComm := TRUE;
   AlmTypeOkShort.SafeEmg := TRUE;
   AlmTypeOkShort.SafeGuards := TRUE;
   AlmTypeOkShort.GtaAirGroup := TRUE;
   AlmTypeOkShort.Major := TRUE;
   AlmTypeOkShort.Minor := TRUE;
   AlmTypeOkShort.Spare07 := TRUE;
   AlmTypeOkShort.Spare08 := TRUE;
   AlmTypeOkShort.Spare09 := TRUE;
   AlmTypeOkShort.Spare10 := TRUE;
   AlmTypeOkShort.Spare11 := TRUE;
   AlmTypeOkShort.Spare12 := TRUE;
   AlmTypeOkShort.Spare13 := TRUE;
   AlmTypeOkShort.Spare14 := TRUE;
   AlmTypeOkShort.Spare15 := TRUE;
   AlmTypeOkShort.Spare16 := TRUE;
   AlmTypeOkShort.Spare17 := TRUE;
   AlmTypeOkShort.Spare18 := TRUE;
   AlmTypeOkShort.Spare19 := TRUE;
   AlmTypeOkShort.Spare20 := TRUE;
   AlmTypeOkShort.Spare21 := TRUE;
   AlmTypeOkShort.Spare22 := TRUE;
   AlmTypeOkShort.Spare23 := TRUE;
   AlmTypeOkShort.Spare24 := TRUE;
   AlmTypeOkShort.Spare25 := TRUE;
   AlmTypeOkShort.Spare26 := TRUE;
   AlmTypeOkShort.Spare27 := TRUE;
   AlmTypeOkShort.Spare28 := TRUE;
   AlmTypeOkShort.Spare29 := TRUE;
   AlmTypeOkShort.Spare30 := TRUE;
   AlmTypeOkShort.Spare31 := TRUE;
   AlmCauseOkShort.Ope := TRUE;
   AlmCauseOkShort.Ust := TRUE;
   AlmCauseOkShort.Dst := TRUE;
   AlmCauseOkShort.Ext := TRUE;
   AlmCauseOkShort.Mac := TRUE;
   AlmCauseOkShort.Spare05 := TRUE;
   AlmCauseOkShort.Spare06 := TRUE;
   AlmCauseOkShort.Spare07 := TRUE;
   AlmCauseOkShort.Spare08 := TRUE;
   AlmCauseOkShort.Spare09 := TRUE;
   AlmCauseOkShort.Spare10 := TRUE;
   AlmCauseOkShort.Spare11 := TRUE;
   AlmCauseOkShort.Spare12 := TRUE;
   AlmCauseOkShort.Spare13 := TRUE;
   AlmCauseOkShort.Spare14 := TRUE;
   AlmCauseOkShort.Spare15 := TRUE;
   AlmCauseOkShort.Spare16 := TRUE;
   AlmCauseOkShort.Spare17 := TRUE;
   AlmCauseOkShort.Spare18 := TRUE;
   AlmCauseOkShort.Spare19 := TRUE;
   AlmCauseOkShort.Spare20 := TRUE;
   AlmCauseOkShort.Spare21 := TRUE;
   AlmCauseOkShort.Spare22 := TRUE;
   AlmCauseOkShort.Spare23 := TRUE;
   AlmCauseOkShort.Spare24 := TRUE;
   AlmCauseOkShort.Spare25 := TRUE;
   AlmCauseOkShort.Spare26 := TRUE;
   AlmCauseOkShort.Spare27 := TRUE;
   AlmCauseOkShort.Spare28 := TRUE;
   AlmCauseOkShort.Spare29 := TRUE;
   AlmCauseOkShort.Spare30 := TRUE;
   AlmCauseOkShort.Spare31 := TRUE;
   AlmStructShort.Category[32..63] := 1;
   AlmStructShort.Category[64..95] := 2;
   AlmStructShort.Category[96..127] := 3;
   AlmStructShort.Category[128..159] := 4;
   AlmStructShort.Category[160..191] := 5;
   AlmStructShort.Category[192..1023] := 6;
   AlmStructShort.BannerPriority[32..63] := 1;
   AlmStructShort.BannerPriority[64..95] := 2;
   AlmStructShort.BannerPriority[96..127] := 3;
   AlmStructShort.BannerPriority[128..159] := 4;
   AlmStructShort.BannerPriority[160..191] := 5;
   AlmStructShort.BannerPriority[192..1023] := 6;
   AlmStructShort.Cause[0..63] := 4;
   AlmStructShort.Cause[128..159] := 3;
   AlmStructShort.Cause[160..1023] := 4;
   AlmBannerFbkShort.AlmPriority := 100;
   AlmBannerFbkShort.AlmCategory := -1;
   AlmBannerFbkShort.AlmCause := -1;
   AlmBannerFbkShort.AlmID := -1;
   // Sign.General."0" : GLOBAL.Sign.General.0 > Circuit breaker protection series not blocking (1PW111)
   // Sign.General."1" : GLOBAL.Sign.General.1 > Overtemperature cabinet door 2 (1PLC360BT2)
   // Sign.General."2" : GLOBAL.Sign.General.2 > Overtemperature cabinet door 4 (1PLC360BT3)
   // Sign.General."3" : GLOBAL.Sign.General.3 > Overtemperature cabinet door 7 (1PLC310BT9)
   // Sign.General."4" : GLOBAL.Sign.General.4
   // Sign.General."5" : GLOBAL.Sign.General.5 > Circuit breaker series lights power supply (1PW115)
   // Sign.General."6" : GLOBAL.Sign.General.6 > Cabinet air conditioning fault
   // Sign.General."7" : GLOBAL.Sign.General.7
   // Sign.General."8" : GLOBAL.Sign.General.8 > Recipe upload to HMI error
   // Sign.General."9" : GLOBAL.Sign.General.9 > Recipe nr.0 active
   // Sign.General."10" : GLOBAL.Sign.General.10 > Recipe not saved
   // Sign.General."11" : GLOBAL.Sign.General.11 > Recipe not loaded
   // Sign.General."12" : GLOBAL.Sign.General.12 > Maintenance configuration recipe upload to HMI error
   // Sign.General."13" : GLOBAL.Sign.General.13 > Totalizers recipe upload to HMI error
   // Sign.General."14" : GLOBAL.Sign.General.14
   Sign.General."15" := TRUE;   // GLOBAL.Sign.General.15 > Downstream packaging disabled from hmi
   // Sign.General."16" : GLOBAL.Sign.General.16 > Downstream packaging not ready
   // Sign.General."17" : GLOBAL.Sign.General.17 > Downstream packaging buffer full
   // Sign.General."18" : GLOBAL.Sign.General.18 > Line Empty
   // Sign.General."19" : GLOBAL.Sign.General.19
   // Sign.General."20" : GLOBAL.Sign.General.20 > Connection HMI client cabinet error
   Sign.General."21" := FALSE;   // GLOBAL.Sign.General.21 > Connection HMI client DP1 error
   Sign.General."22" := FALSE;   // GLOBAL.Sign.General.22 > Connection HMI client DP2 error
   Sign.General."23" := FALSE;   // GLOBAL.Sign.General.23 > Connection HMI client DP3 error
   Sign.General."24" := FALSE;   // GLOBAL.Sign.General.24 > Connection HMI client DP4 error
   // Sign.General."25" : GLOBAL.Sign.General.25 > Connection HMI client RD1 error
   // Sign.General."26" : GLOBAL.Sign.General.26
   // Sign.General."27" : GLOBAL.Sign.General.27
   // Sign.General."28" : GLOBAL.Sign.General.28
   // Sign.General."29" : GLOBAL.Sign.General.29
   // Sign.General."30" : GLOBAL.Sign.General.30
   // Sign.General."31" : GLOBAL.Sign.General.31
   SignStruct.Sign[0] := 32768;
   SignStruct.BannerPriority[7..11] := 3;
   SignStruct.BannerPriority[13..14] := 3;
   SignStruct.BannerPriority[18..31] := 3;
   SignBannerFbk.SignID := 645015;
   Input.BrkPwr1 := TRUE;
   Input.BrkPwr2 := TRUE;
   Input.BrkSrsLgh := TRUE;
   Input.BrkSrsCab := TRUE;
   Input.BrkGenCab := TRUE;
   Input.BrkSrsBlk := TRUE;
   Input.BrkSrsBlkDep := TRUE;
   Input.BrkSrsNotBlk := TRUE;
   Input.BrkSrsSin := TRUE;
   Input.BrkSrsFld := TRUE;
   Input.BrkSrsVlv := TRUE;
   Input.DisPwr := TRUE;
   Input.AirOkGta1 := TRUE;
   Input.AirOkGta2 := TRUE;
   Input.AirOkGta3 := TRUE;
   Input.AirOkGta4 := FALSE;
   Input.AirOkGta5 := FALSE;
   Input.Prs24Vdc := TRUE;
   Input.Safety.GtaZon4_ModIstFlt := TRUE;
   Input.Safety.FbkPwrCntIH1 := TRUE;
   Input.Safety.FbkPwrCntCM1 := TRUE;
   Input.Safety.SimPwrOn := TRUE;
   Output.CmdPwrShort := 8191;
   Output.CmdPwrLong := 8191;
   Ons.CmdPwrShort := FALSE;
   Ons.CmdPwrLong := FALSE;
   Ons.PidCounter := FALSE;
   Ons.EthModCounter := FALSE;
   AirTreatment.AlmOk := TRUE;
   AirTreatment.CycleActivated := TRUE;
   AirTreatment.CycleOn := TRUE;
   AirTreatment.Output.GrnLgh := TRUE;
   AirTreatment.TON_Defrost.PT := T#45M;
   AirTreatment.TON_StopBtn.PT := T#5S;
   Summ.PresAlm := TRUE;
   Summ.PresSign := TRUE;
   Summ.AbortAlmOk := FALSE;
   Summ.Aborted := TRUE;
   Summ.Ena_Suspended := TRUE;
   Summ.ManSel := TRUE;
   Summ.ManSelModulesSelected := TRUE;
   Summ.AlmOk.ThSwitch := TRUE;
   Summ.AlmOk.SafeComm := TRUE;
   Summ.AlmOk.SafeEmg := TRUE;
   Summ.AlmOk.SafeGuards := FALSE;
   Summ.AlmOk.GtaAirGroup := FALSE;
   Summ.AlmOk.Major := TRUE;
   Summ.AlmCauseOk.Ope := FALSE;
   Summ.AlmCauseOk.Ust := TRUE;
   Summ.AlmCauseOk.Dst := TRUE;
   Summ.AlmCauseOk.Ext := FALSE;
   LightSiren.Cfg_RstPbt := -1;
   LightSiren.Cfg_Siren := 1;
   LightSiren.Cfg_Stack := 1;
   LightSiren.Frequency1.RstPbtLgh := TRUE;
   LightSiren.Frequency1.YelStkLgh := TRUE;
   LightSiren.Frequency1.Cust1_RstPbtLgh := TRUE;
   LightSiren.Frequency1.Cust1_RedStkLgh := TRUE;
   ExchangeCmd.Communication.RunMode := TRUE;
   ExchangeCmd.Gen.RecipeMngByHmi := TRUE;
   ExchangeCmd.Gen.PwrDrv := TRUE;
   ExchangeCmd.Gen.Downstream_RunEnable := TRUE;
   ExchangeCmd.Gen.AirCycleOn := TRUE;
   ExchangeCmd.Gen.SelSetpointAirTreatment := TRUE;
   ExchangeCmd.Gen.CopyHmiToWorkEna := TRUE;
   ExchangeCmd.Gen.CfgPbtAutoShort := 65535;
   ExchangeCmd.Gen.CfgPbtAutoLong := 65535;
   ExchangeCmd.Gen.CfgPbtManLong := 65535;
   ExchangeCmd.Summ.AbortAlmOk := FALSE;
   ExchangeCmd.Summ.Ena_Suspended := TRUE;
   ExchangeCmd.Clock._0_0166Hz := TRUE;
   ExchangeCmd.Clock._0_5Hz := TRUE;
   ExchangeCmd.Clock._1Hz := TRUE;
   ExchangeCmd.Clock._2Hz := FALSE;
   ExchangeCmd.Clock._2_5Hz := FALSE;
   ExchangeCmd.Clock._5Hz := FALSE;
   ExchangeCmd.Clock._10Hz := TRUE;
   ExchangeCmd.HmiVisAlmTypeBool.SafeGuards := TRUE;
   ExchangeCmd.HmiVisAlmTypeBool.GtaAirGroup := FALSE;
   ExchangeCmd.HmiVisAlmTypeBool.Minor := FALSE;
   ExchangeCmd.Panel[1].ConnectionCheck := TRUE;
   ExchangeCmd.Panel[4].ConnectionCheck := TRUE;
   ExchangeCmd.Panel[0..4].ScreenNumber := 0;
   ExchangeCmd.Panel[5].ScreenNumber := 332_030_302;
   ExchangeCmd.Panel[6].ScreenNumber := -1;
   ExchangeCmd."DeviceDiagCab&Field"[0] := TRUE;
   ExchangeCmd."DeviceDiagCab&Field"[8..9] := TRUE;
   ExchangeCmd."DeviceDiagCab&Field"[15..18] := TRUE;
   ExchangeCmd."DeviceDiagCab&Field"[21..22] := TRUE;
   ExchangeCmd."DeviceDiagCab&Field"[25..26] := TRUE;
   ExchangeCmd."DeviceDiagCab&Field"[29..50] := TRUE;
   ExchangeCmd."DeviceDiagCab&Field"[61..64] := TRUE;
   ExchangeCmd."DeviceDiagCab&Field"[66..68] := TRUE;
   ExchangeCmd."DeviceDiagCab&Field"[70..72] := TRUE;
   ExchangeCmd."DeviceDiagCab&Field"[74] := TRUE;
   ExchangeCmd."DeviceDiagCab&Field"[76..77] := TRUE;
   ExchangeCmd."DeviceDiagCab&Field"[79..80] := TRUE;
   ExchangeCmd."DeviceDiagCab&Field"[83..85] := TRUE;
   ExchangeCmd.RecipeNumOnline := 4;
   ExchangeCmd.RecipeNumOffline := 15;
   ExchangeCmd.ReqDeviceDiag := 5;
   ExchangeCmd.ReqInverterDiag := 18;
   ExchangeCmd.StrobePID := 128;
   ExchangeCmd.SwitchboardsNumber := 16;
   ExchangeCmd.PanelsNumber := 7;
   ExchangeCmd.TimePIDexecution := 8.0;
   ExchangeCmd.TimeCurrent := 1_727_980_997_860_936;
   ExchangeCmd_Switchboard.Communication.RunMode := TRUE;
   ExchangeCmd_Switchboard.LightSiren[0..15].RstPbtLgh := TRUE;
   ExchangeCmd_Switchboard.LightSiren[0].YelStkLgh := TRUE;
   ExchangeCmd_Switchboard.LightSiren[0].BluStkLgh := FALSE;
   ExchangeCmd_Switchboard.LightSiren[3].BluStkLgh := FALSE;
   ExchangeCmd_Switchboard.LightSiren[0..15].Cust1_RstPbtLgh := TRUE;
   ExchangeCmd_Switchboard.LightSiren[0].Cust1_RedStkLgh := TRUE;
   ExchangeCmd_Switchboard.LightSiren[0].Cust1_BluStkLgh := FALSE;
   ExchangeCmd_Switchboard.LightSiren[3].Cust1_BluStkLgh := FALSE;
   Downstream.RunEnable := TRUE;
   Downstream.PresReject := TRUE;
   Downstream.TON_DelayRun.PT := T#2S;
   Downstream.TON_DelayRun.ET := T#2S;
   Downstream.TON_DelayRun.IN := TRUE;
   Downstream.TON_DelayRun.Q := TRUE;
   Downstream.TON_DelayWatchdogOn.PT := T#5S;
   Downstream.TON_DelayWatchdogOff.PT := T#5S;
   Downstream.TON_BufferAlm.PT := T#5S;
   "MyStateDeviceCab&Field"[0] := TRUE;
   "MyStateDeviceCab&Field"[8..9] := TRUE;
   "MyStateDeviceCab&Field"[15..18] := TRUE;
   "MyStateDeviceCab&Field"[21..22] := TRUE;
   "MyStateDeviceCab&Field"[25..26] := TRUE;
   "MyStateDeviceCab&Field"[29..50] := TRUE;
   "MyStateDeviceCab&Field"[61..64] := TRUE;
   "MyStateDeviceCab&Field"[66..68] := TRUE;
   "MyStateDeviceCab&Field"[70..72] := TRUE;
   "MyStateDeviceCab&Field"[74] := TRUE;
   "MyStateDeviceCab&Field"[76..77] := TRUE;
   "MyStateDeviceCab&Field"[79..80] := TRUE;
   "MyStateDeviceCab&Field"[83..85] := TRUE;
   DC_Bus_Converter1.FBK.BusReadyStatus := TRUE;
   DC_Bus_Converter2.FBK.BusReadyStatus := TRUE;
   DC_Bus_Converter3.FBK.BusReadyStatus := TRUE;
END_DATA_BLOCK
